// TIA Portal V20 export
TYPE "typeSequenceControlNodeJobInterface_topTapeAttachment"
// stored: Namespace Unit1.Em3
   STRUCT
      tapeGetJob2 : "LER_typeJobInterface";
      tape1PutJob3 : "LER_typeJobInterface";
      tape2PutJob4 : "LER_typeJobInterface";
      tapeIdleJob5 { S7_SetPoint := 'True'} : "LER_typeJobInterface";
   END_STRUCT;
END_TYPE
